FUNCTION_BLOCK automaton
  (* Standard: 61499-2 *)
  (* Version 0.0, 2020-05-11, fbSAT, nxtControl GmbH *)
  PACKAGE Main;
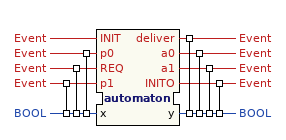
  EVENT_INPUT
    INIT;
    p0 WITH x;
    REQ WITH x;
    p1 WITH x;
  END_EVENT
  EVENT_OUTPUT
    deliver WITH y;
    a0 WITH y;
    a1 WITH y;
    INITO WITH y;
  END_EVENT
  VAR_INPUT
    x : BOOL;
  END_VAR
  VAR_OUTPUT
    y : BOOL;
  END_VAR
  EC_STATES
    START;
    INIT : INIT -> INITO;
    s1 : s1_0_0;
    s2 : s2_0_0 -> deliver;
    s3 : s3_0_0 -> a0;
    s4 : s4_0_0 -> deliver;
    s5 : s5_0_0 -> a1;
  END_STATES
  EC_TRANSITIONS
    START TO INIT := INIT;
    INIT TO s1 := 1;
    s1 TO s2 := p0&NOT x;
    s2 TO s3 := REQ&NOT x;
    s3 TO s4 := p1&NOT x;
    s4 TO s5 := REQ&NOT x;
    s5 TO s2 := p0&NOT x;
  END_TRANSITIONS
  ALGORITHM INIT IN ST:
y:=FALSE;
  END_ALGORITHM
  ALGORITHM s2_0_0 IN ST:
y:=FALSE;
  END_ALGORITHM
  ALGORITHM s3_0_0 IN ST:
y:=FALSE;
  END_ALGORITHM
  ALGORITHM s4_0_0 IN ST:
y:=FALSE;
  END_ALGORITHM
  ALGORITHM s5_0_0 IN ST:
y:=FALSE;
  END_ALGORITHM
END_FUNCTION_BLOCK
